// TwinCAT 3 PLC project PLC_1
// ProgramVersion: 3.1.4023.0
// libraries:
//   Tc2_Standard, * (Beckhoff Automation GmbH)
//   Tc2_System, * (Beckhoff Automation GmbH)
//   Tc2_Utilities, * (Beckhoff Automation GmbH)
//   Tc3_IotBase, * (Beckhoff Automation GmbH)
//   Tc3_JsonXml, * (Beckhoff Automation GmbH)
//   Tc3_Module, * (Beckhoff Automation GmbH)
// project tree:
//   / PlcTask.TcTTO
//   POUs/ FB_HttpPut.TcPOU, MAIN.TcPOU

CONFIGURATION PLC_1
    RESOURCE PLC ON TwinCAT3
        TASK PlcTask(INTERVAL := T#50us, PRIORITY := 20);
        PROGRAM MAIN WITH PlcTask : MAIN;
    END_RESOURCE
END_CONFIGURATION

// ---- POUs/MAIN.TcPOU
PROGRAM MAIN
VAR
	bPut: BOOL;
	fbHttpClient: FB_IotHttpClient := (sHostName:= '192.168.1.99',bKeepAlive := TRUE, tConnectionTimeout:=T#10S);
	fbPut: FB_HttpPut;
	bBlinkingMode: BOOL;
	fbTimer: ton := (pt:=T#500MS);
	nColor: UINT;
END_VAR

IF NOT fbHttpClient.bConfigured THEN
	fbHttpClient.nHostPort := 80;
	fbHttpClient.stTLS.bNoServerCertCheck:= TRUE;
END_IF

IF fbHttpClient.bConfigured THEN
	fbPut(bSend := bPut, fbClient:= fbHttpClient, nColor:= nColor);
END_IF

IF bBlinkingMode THEN
	fbTimer(in:= NOT fbTimer.Q);
	IF fbTimer.Q THEN
		nColor:=nColor+5000;
        IF nColor=65000 THEN
            nColor:=0;
        END_IF
		IF bPut THEN
			bPut:= FALSE;
		ELSE
			bPut:= TRUE;
		END_IF
	END_IF
END_IF

fbHttpClient.Execute();

END_PROGRAM

// ---- POUs/FB_HttpPut.TcPOU
FUNCTION_BLOCK FB_HttpPut
VAR_INPUT
	bSend                : BOOL;
    nColor               : UINT;
END_VAR
VAR_IN_OUT
	fbClient             : FB_IotHttpClient;
END_VAR
VAR_OUTPUT
	bBusy                : BOOL;
    bError               : BOOL;
END_VAR
VAR
	fbRequest: FB_IotHttpRequest;
	fbJson: FB_JsonDomParser;
	fbJsonWriter: FB_JsonSaxWriter;
	nState: UDINT;
	RisingEdge: R_TRIG;
	
	sContent: STRING(511);
	sSend: STRING(511);
	
	jsonDoc: SJsonValue;
	jsonVal: SJsonValue;
	sResultValue: STRING;

END_VAR

RisingEdge(clk:= bSend);

CASE nState OF
0: 
	fbJsonWriter.StartObject();
	fbJsonWriter.AddKey('sat');
	fbJsonWriter.AddUdint(254);
	fbJsonWriter.AddKey('bri');
	fbJsonWriter.AddUdint(200);
	fbJsonWriter.AddKey('hue');
	fbJsonWriter.AddUdint(nColor);
	fbJsonWriter.AddKey('transitiontime');
	fbJsonWriter.AddUdint(1);
	fbJsonWriter.EndObject();
	sSend:= fbJsonWriter.GetDocument();
	fbJsonWriter.ResetDocument();
	
	IF RisingEdge.Q THEN
		IF fbRequest.SendRequest(sUri:='/api/OOrb8w4GpeITNRtK0w5Yf6Ke3p1k6PnnwycVn68a/lights/4/state', fbClient:=fbClient, eRequestType:= ETcIotHttpRequestType.HTTP_PUT,
			pContent:= ADR(sSend), nContentSize:= LEN2(ADR(sSend)), 0) THEN
			
			nState:= 1;
			bBusy:= TRUE;
			bError:= FALSE;
		END_IF
	END_IF
	
1:
	IF NOT fbRequest.bBusy THEN
		bError:= TRUE;
		IF NOT fbRequest.bError THEN
			fbRequest.GetContent(pContent:= ADR(sContent), nContentSize:= SIZEOF(sContent), bSetNullTermination:= TRUE);
			IF fbRequest.nStatusCode >= 200 AND fbRequest.nStatusCode < 300 THEN              
                bError:= FALSE;    
            END_IF
        END_IF
        nState:= 0;
        bBusy:= FALSE;
	END_IF
END_CASE

END_FUNCTION_BLOCK
